// TIA Portal V20 export
DATA_BLOCK "IDB_OPC_Communication"   // DB42
// stored: InstanceOfName ProductionLine.FB_OPC_Communication, InstanceOfType FB, Namespace ProductionLine
"ProductionLine.FB_OPC_Communication"
   // VAR
   //    Communication_DP1 : "ProductionLine.FB_OPC_DestRequest";
   //    Communication_DP2 : "ProductionLine.FB_OPC_DestRequest";
   //    Communication_DP3 : "ProductionLine.FB_OPC_DestRequest";
   //    Communication_DP4 : "ProductionLine.FB_OPC_DestRequest";
   //    Communication_IP1 : "ProductionLine.FB_OPC_DestInfo";
   //    Communication_IP2 : "ProductionLine.FB_OPC_DestInfo";
   //    Communication_IP3 : "ProductionLine.FB_OPC_DestInfo";
   //    Communication_IP4 : "ProductionLine.FB_OPC_DestInfo";
   //    Communication_IP5 : "ProductionLine.FB_OPC_DestInfo";
   //    Communication_IP6 : "ProductionLine.FB_OPC_DestInfo";
   //    Communication_IP7 : "ProductionLine.FB_OPC_DestInfo";
   //    Communication_IP8 : "ProductionLine.FB_OPC_DestInfo";
   //    Communication_IP9 : "ProductionLine.FB_OPC_DestInfo";
   //    Communication_SYS_OP : "ProductionLine.FB_OPC_SysStatus";
   //    Communication_SYS_OP_Source { S7_SetPoint := 'True'} : "ProductionLine.OPC_SystemStatus";
   //    Communication_SYS_OP_Ack { S7_SetPoint := 'True'} : "ProductionLine.OPC_SystStatus_Ack";
   //    timPeriodicSend { S7_SetPoint := 'True'} : IEC_TIMER;
   //    timWatchdog { S7_SetPoint := 'True'} : IEC_TIMER;
   //    Communication_fault : Bool;
   // END_VAR
BEGIN
END_DATA_BLOCK
